Fanuc KAREL source: SET_STR_REG.kl

PROGRAM T
%NOLOCKGROUP
VAR
 v0 : INTEGER
 v1 : STRING[40]
 v2 : INTEGER
BEGIN
 SET_STR_REG(v0, v1, v2)
END T
